FUNCTION_BLOCK fb_mapping
VAR_INPUT
END_VAR
VAR_OUTPUT
END_VAR
VAR
	fbi_ejector_io: ARRAY[1..3] OF fb_ejector_io;
	fbi_sv_io: ARRAY[1..8] OF  fb_sv_io;
	fbi_ele_io: ARRAY[1..6] OF  fb_ele_io;
END_VAR

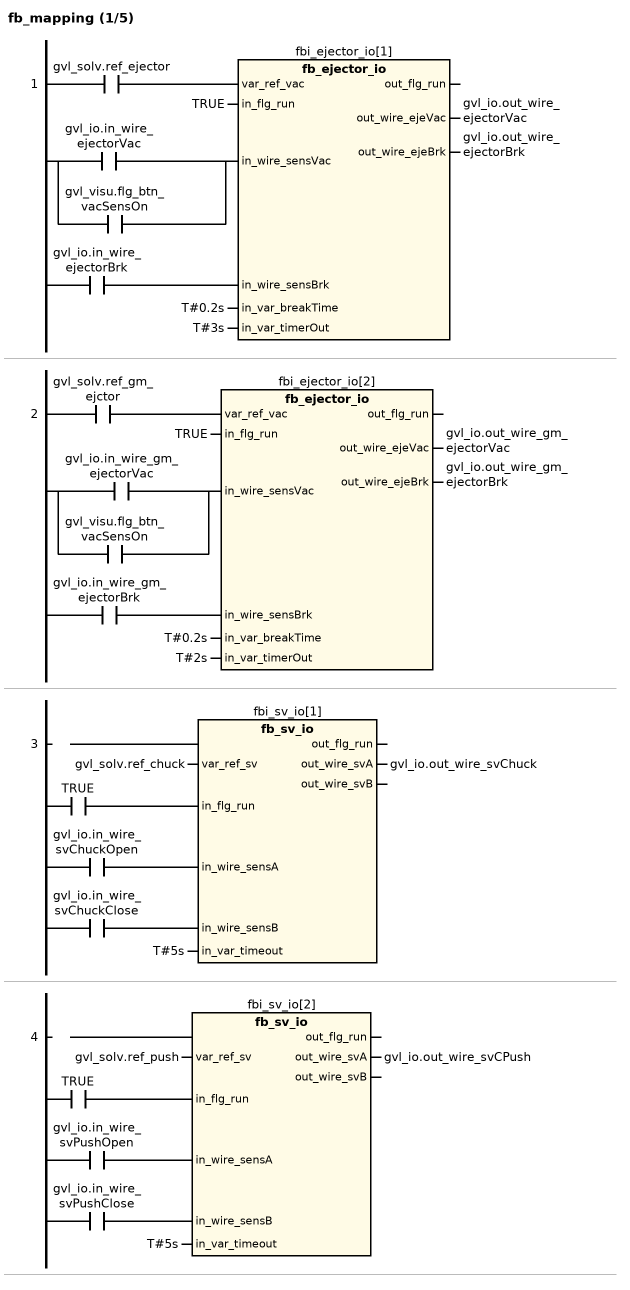
// NETWORK 1
fbi_ejector_io[1](
    var_ref_vac := gvl_solv.ref_ejector,
    in_flg_run := TRUE,
    in_wire_sensVac := gvl_io.in_wire_ejectorVac OR gvl_visu.flg_btn_vacSensOn,
    in_wire_sensBrk := gvl_io.in_wire_ejectorBrk,
    in_var_breakTime := T#0.2s,
    in_var_timerOut := T#3s,
    out_wire_ejeVac => gvl_io.out_wire_ejectorVac,
    out_wire_ejeBrk => gvl_io.out_wire_ejectorBrk); // fb_ejector_io

// NETWORK 2
fbi_ejector_io[2](
    var_ref_vac := gvl_solv.ref_gm_ejctor,
    in_flg_run := TRUE,
    in_wire_sensVac := gvl_io.in_wire_gm_ejectorVac OR gvl_visu.flg_btn_vacSensOn,
    in_wire_sensBrk := gvl_io.in_wire_gm_ejectorBrk,
    in_var_breakTime := T#0.2s,
    in_var_timerOut := T#2s,
    out_wire_ejeVac => gvl_io.out_wire_gm_ejectorVac,
    out_wire_ejeBrk => gvl_io.out_wire_gm_ejectorBrk); // fb_ejector_io

// NETWORK 3
fbi_sv_io[1](
    var_ref_sv := gvl_solv.ref_chuck,
    in_flg_run := TRUE,
    in_wire_sensA := gvl_io.in_wire_svChuckOpen,
    in_wire_sensB := gvl_io.in_wire_svChuckClose,
    in_var_timeout := T#5s,
    out_wire_svA => gvl_io.out_wire_svChuck); // fb_sv_io

// NETWORK 4
fbi_sv_io[2](
    var_ref_sv := gvl_solv.ref_push,
    in_flg_run := TRUE,
    in_wire_sensA := gvl_io.in_wire_svPushOpen,
    in_wire_sensB := gvl_io.in_wire_svPushClose,
    in_var_timeout := T#5s,
    out_wire_svA => gvl_io.out_wire_svCPush); // fb_sv_io

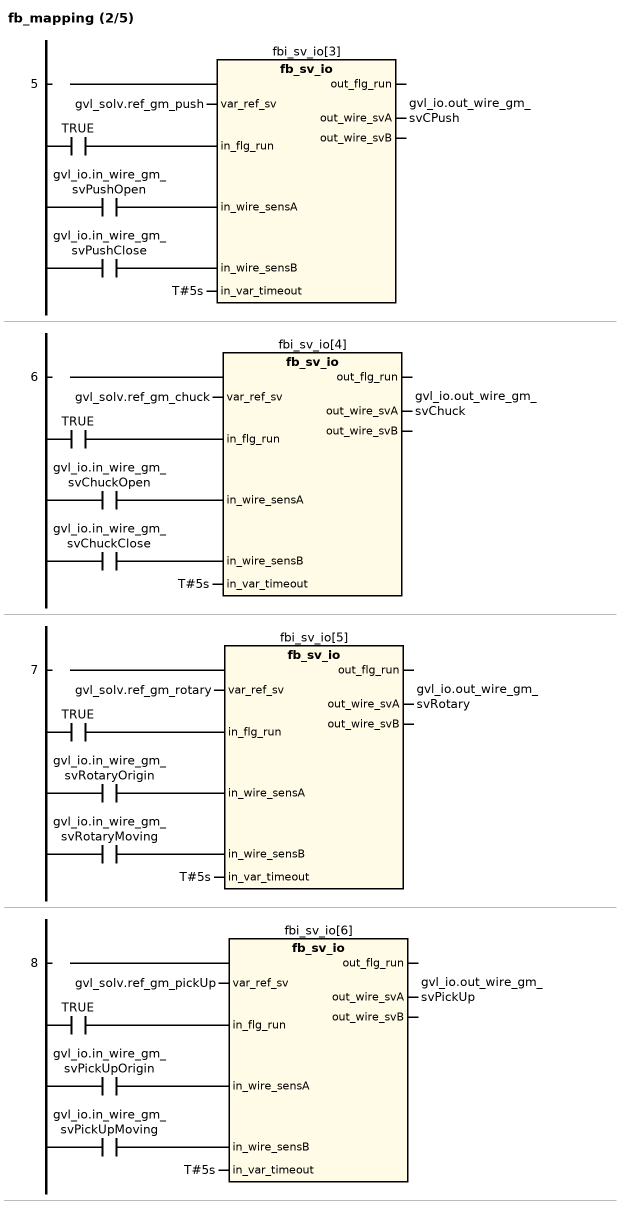
// NETWORK 5
fbi_sv_io[3](
    var_ref_sv := gvl_solv.ref_gm_push,
    in_flg_run := TRUE,
    in_wire_sensA := gvl_io.in_wire_gm_svPushOpen,
    in_wire_sensB := gvl_io.in_wire_gm_svPushClose,
    in_var_timeout := T#5s,
    out_wire_svA => gvl_io.out_wire_gm_svCPush); // fb_sv_io

// NETWORK 6
fbi_sv_io[4](
    var_ref_sv := gvl_solv.ref_gm_chuck,
    in_flg_run := TRUE,
    in_wire_sensA := gvl_io.in_wire_gm_svChuckOpen,
    in_wire_sensB := gvl_io.in_wire_gm_svChuckClose,
    in_var_timeout := T#5s,
    out_wire_svA => gvl_io.out_wire_gm_svChuck); // fb_sv_io

// NETWORK 7
fbi_sv_io[5](
    var_ref_sv := gvl_solv.ref_gm_rotary,
    in_flg_run := TRUE,
    in_wire_sensA := gvl_io.in_wire_gm_svRotaryOrigin,
    in_wire_sensB := gvl_io.in_wire_gm_svRotaryMoving,
    in_var_timeout := T#5s,
    out_wire_svA => gvl_io.out_wire_gm_svRotary); // fb_sv_io

// NETWORK 8
fbi_sv_io[6](
    var_ref_sv := gvl_solv.ref_gm_pickUp,
    in_flg_run := TRUE,
    in_wire_sensA := gvl_io.in_wire_gm_svPickUpOrigin,
    in_wire_sensB := gvl_io.in_wire_gm_svPickUpMoving,
    in_var_timeout := T#5s,
    out_wire_svA => gvl_io.out_wire_gm_svPickUp); // fb_sv_io

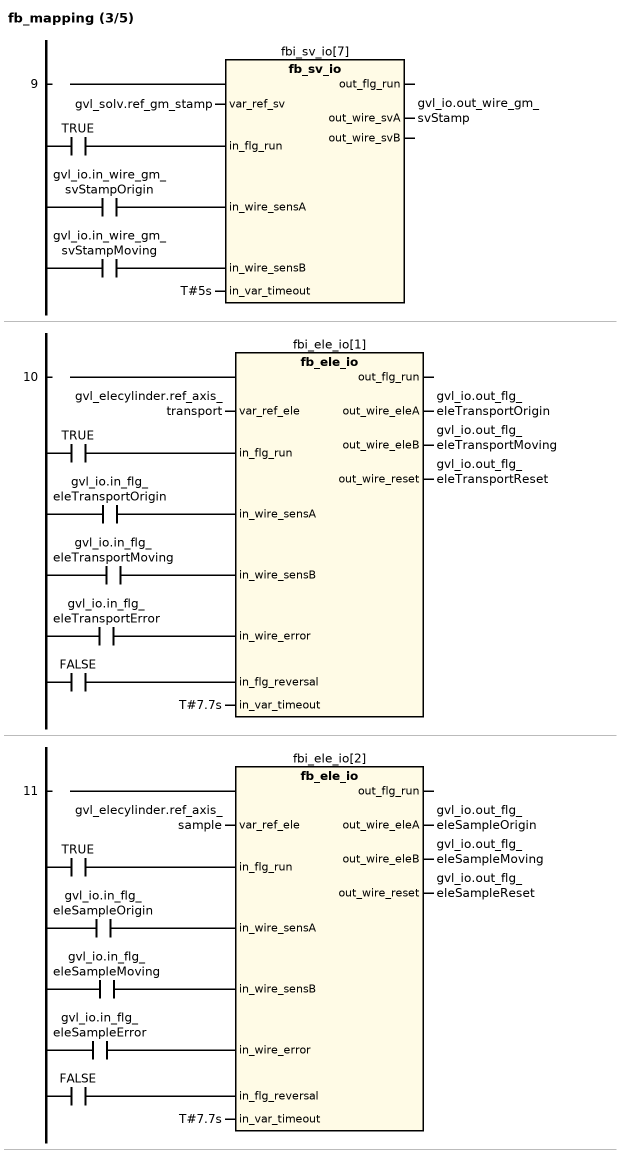
// NETWORK 9
fbi_sv_io[7](
    var_ref_sv := gvl_solv.ref_gm_stamp,
    in_flg_run := TRUE,
    in_wire_sensA := gvl_io.in_wire_gm_svStampOrigin,
    in_wire_sensB := gvl_io.in_wire_gm_svStampMoving,
    in_var_timeout := T#5s,
    out_wire_svA => gvl_io.out_wire_gm_svStamp); // fb_sv_io

// NETWORK 10
fbi_ele_io[1](
    var_ref_ele := gvl_elecylinder.ref_axis_transport,
    in_flg_run := TRUE,
    in_wire_sensA := gvl_io.in_flg_eleTransportOrigin,
    in_wire_sensB := gvl_io.in_flg_eleTransportMoving,
    in_wire_error := gvl_io.in_flg_eleTransportError,
    in_flg_reversal := FALSE,
    in_var_timeout := T#7.7s,
    out_wire_eleA => gvl_io.out_flg_eleTransportOrigin,
    out_wire_eleB => gvl_io.out_flg_eleTransportMoving,
    out_wire_reset => gvl_io.out_flg_eleTransportReset); // fb_ele_io

// NETWORK 11
fbi_ele_io[2](
    var_ref_ele := gvl_elecylinder.ref_axis_sample,
    in_flg_run := TRUE,
    in_wire_sensA := gvl_io.in_flg_eleSampleOrigin,
    in_wire_sensB := gvl_io.in_flg_eleSampleMoving,
    in_wire_error := gvl_io.in_flg_eleSampleError,
    in_flg_reversal := FALSE,
    in_var_timeout := T#7.7s,
    out_wire_eleA => gvl_io.out_flg_eleSampleOrigin,
    out_wire_eleB => gvl_io.out_flg_eleSampleMoving,
    out_wire_reset => gvl_io.out_flg_eleSampleReset); // fb_ele_io

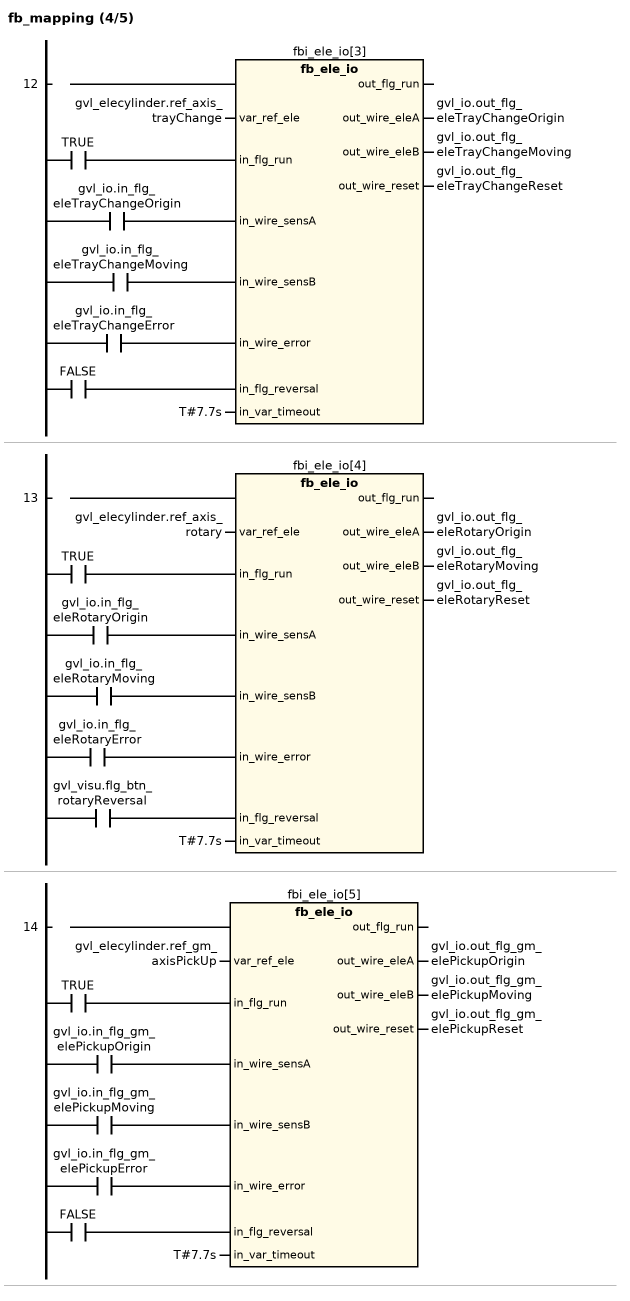
// NETWORK 12
fbi_ele_io[3](
    var_ref_ele := gvl_elecylinder.ref_axis_trayChange,
    in_flg_run := TRUE,
    in_wire_sensA := gvl_io.in_flg_eleTrayChangeOrigin,
    in_wire_sensB := gvl_io.in_flg_eleTrayChangeMoving,
    in_wire_error := gvl_io.in_flg_eleTrayChangeError,
    in_flg_reversal := FALSE,
    in_var_timeout := T#7.7s,
    out_wire_eleA => gvl_io.out_flg_eleTrayChangeOrigin,
    out_wire_eleB => gvl_io.out_flg_eleTrayChangeMoving,
    out_wire_reset => gvl_io.out_flg_eleTrayChangeReset); // fb_ele_io

// NETWORK 13
fbi_ele_io[4](
    var_ref_ele := gvl_elecylinder.ref_axis_rotary,
    in_flg_run := TRUE,
    in_wire_sensA := gvl_io.in_flg_eleRotaryOrigin,
    in_wire_sensB := gvl_io.in_flg_eleRotaryMoving,
    in_wire_error := gvl_io.in_flg_eleRotaryError,
    in_flg_reversal := gvl_visu.flg_btn_rotaryReversal,
    in_var_timeout := T#7.7s,
    out_wire_eleA => gvl_io.out_flg_eleRotaryOrigin,
    out_wire_eleB => gvl_io.out_flg_eleRotaryMoving,
    out_wire_reset => gvl_io.out_flg_eleRotaryReset); // fb_ele_io

// NETWORK 14
fbi_ele_io[5](
    var_ref_ele := gvl_elecylinder.ref_gm_axisPickUp,
    in_flg_run := TRUE,
    in_wire_sensA := gvl_io.in_flg_gm_elePickupOrigin,
    in_wire_sensB := gvl_io.in_flg_gm_elePickupMoving,
    in_wire_error := gvl_io.in_flg_gm_elePickupError,
    in_flg_reversal := FALSE,
    in_var_timeout := T#7.7s,
    out_wire_eleA => gvl_io.out_flg_gm_elePickupOrigin,
    out_wire_eleB => gvl_io.out_flg_gm_elePickupMoving,
    out_wire_reset => gvl_io.out_flg_gm_elePickupReset); // fb_ele_io

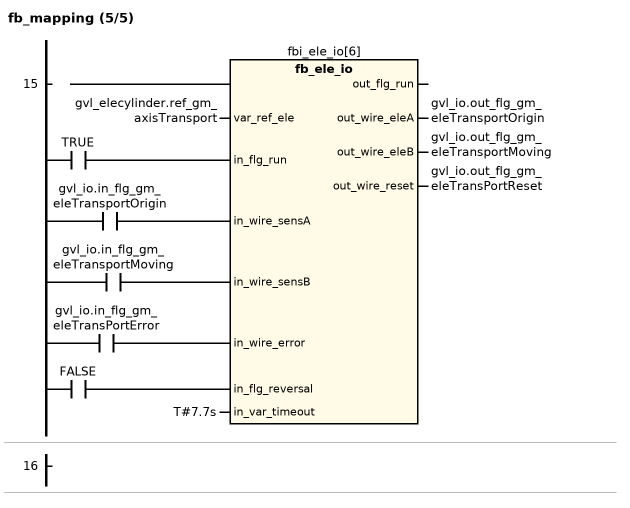
// NETWORK 15
fbi_ele_io[6](
    var_ref_ele := gvl_elecylinder.ref_gm_axisTransport,
    in_flg_run := TRUE,
    in_wire_sensA := gvl_io.in_flg_gm_eleTransportOrigin,
    in_wire_sensB := gvl_io.in_flg_gm_eleTransportMoving,
    in_wire_error := gvl_io.in_flg_gm_eleTransPortError,
    in_flg_reversal := FALSE,
    in_var_timeout := T#7.7s,
    out_wire_eleA => gvl_io.out_flg_gm_eleTransportOrigin,
    out_wire_eleB => gvl_io.out_flg_gm_eleTransportMoving,
    out_wire_reset => gvl_io.out_flg_gm_eleTransPortReset); // fb_ele_io

// NETWORK 16

END_FUNCTION_BLOCK

(* stored: Version 1.1.0.1, ProductVersion 3.1.4024.11
   POU fb_mapping: Id {83adaf20-f572-416c-bb16-5d23cb9a942b}, SpecialFunc None *)
